// TIA Portal V17 export
// export: Created 2025-01-08T13:55:36.5393267Z, ExportSetting WithDefaults, DisplayName Totally Integrated Automation Portal, DisplayVersion V17, DisplayName TIA Portal Openness, DisplayVersion V17, DisplayName TIA Portal Version Control Interface, DisplayVersion V17, DisplayName SINAMICS Startdrive Advanced, DisplayVersion V17 Update2, DisplayName SINAMICS Startdrive G130, G150, S120, S150, SINAMICS MV, S210, DisplayVersion V17 Update2, DisplayName SINAMICS Startdrive G110M, G120, G120C, G120D, G120P, G115D, DisplayVersion V17 Update2, DisplayName STEP 7 Professional, DisplayVersion V17, DisplayName STEP 7 Safety, DisplayVersion V17, DisplayName WinCC Advanced, DisplayVersion V17
TYPE "typeFromHMI"
// stored: IsFailsafeCompliant false
   STRUCT
      xBtn_Stop : Bool;   // Stop HSM
      xBtn_Run : Bool;   // Start HSM
      xBtn_Teach : Bool;   // Calibrate label process = 1
      xBtn_Feed : Bool;   // Feed label manually
      xBtn_Get_FW_MAC : Bool;   // Get firmware version and MAC address.
      xBtn_Activate_Splice : Bool;
      xSend_Para : Bool;
      rLabel_Speed : Real := 60.0;   // Label speed
      xBtn_Save_Par : Bool;   // Save parameters to HSM
      xHSM_Active : Bool := true;   // Enabled = 1, Disabled = 0
      xGet_Parameters : Bool;
      iLabels_Per_Trigger : Int := 1;
      iTrigger_Supression : Int := 0;
      iProduct_Sensor_Polarity : Int := 3;
      iDouble_Label : Int := 0;
      iSpeed_Int_Ext : Int;
      iLabel_Length : Int := 0;
      rLabel_Position : Real := 1.0;   // Calibration offset label position on peeler plate.
      rTrig_Delay : Real := 0.0;   // Delay trigger labelling when sensor trig.
      rSpeed_Offset : Real := 0.0;   // Label speed + speed offset = speed internal
      rGap_Sensor_To_Dispenser_Tongue : Real := 240.0;
      rLabel_Spacing : Real := 2.0;
      rPre_Dispensing_Lenght : Real := 0.0;
      rLabel_Gap : Real := 0.0;
      rSpeed_Offset_Percentage : Real := 0.0;
      ConfigAndMachineParaMask : "HSMConfigAndMachineParameterMask";
   END_STRUCT;
END_TYPE
